// TwinCAT 3 PLC project POS_Temp_system
// ProgramVersion: 3.1.4022.3
// libraries:
//   CAA Types Extern, * (CAA Technical Workgroup)
//   Tc2_ControllerToolbox, * (Beckhoff Automation GmbH)
//   Tc2_Standard, * (Beckhoff Automation GmbH)
//   Tc2_System, * (Beckhoff Automation GmbH)
//   Tc2_Utilities, * (Beckhoff Automation GmbH)
//   Tc3_Module, * (Beckhoff Automation GmbH)
//   VisuSymbols,3.5.10.0,System
// project tree:
//   DUTs/ SeqState.TcTLEO
//   fbBLOCKS/ fbSensorNoise.TcPOU, FirstOrder.TcPOU
//   / GlobalTextList.TcGTLO, PlcTask.TcTTO, Visualization Manager.TcVMO (not stored)
//   GVLs/ GVL_IO.TcGVL
//   POUs/ fBDISCRETE_PID.TcPOU, MAIN.TcPOU
//   PROCESSES/ HEATER_PROCESS.TcPOU, SERVO_POS.TcPOU, TANKLEVEL.TcPOU
//   VISUs/ UserInterface.TcVIS
// real-time tasks:
//   TASK PlcTask: cycle T#10ms, priority 6, ADS port 350
//   TASK VISU_TASK: cycle T#200000us, priority 30, ADS port 351

CONFIGURATION POS_Temp_system
    RESOURCE PLC ON TwinCAT3
        TASK PlcTask(INTERVAL := T#10ms, PRIORITY := 6);
        PROGRAM MAIN WITH PlcTask : MAIN;
        PROGRAM SERVO_POS WITH PlcTask : SERVO_POS;
        PROGRAM HEATER_PROCESS WITH PlcTask : HEATER_PROCESS;
        PROGRAM TANKLEVEL WITH PlcTask : TANKLEVEL;
    END_RESOURCE
END_CONFIGURATION

// ---- DUTs/SeqState.TcTLEO
{attribute 'qualified_only'}
{attribute 'strict'}
TYPE SeqState :
(
	Ready,
	Fill_A,
	Fill_B,
	Heating,
	ToUnload,
	MovingToDrain,
	MovingToStart,
	Drain_1,
	Drain_2
	);
END_TYPE

// ---- GVLs/GVL_IO.TcGVL
{attribute 'qualified_only'}
VAR_GLOBAL
// Process parameters, variables	
	SetPoint_ServoX           :REAL;      // SetPoint X - axis
	SetPointHeater            :REAL;      // SetPoint Heater
	Output_ServoX             :REAL;      // X-axis Position
	Output_Heater             :REAL;      // Temperature Heater
	TankLevelSensor           :REAL;      // Tanklevel analogue sensor 
	ValveA, ValveB, ValveC    :BOOL;      // Valves
	xPushButton1              :BOOL;      // Used for test purposes 
	xPushButton2              :BOOL;      // Used for test purposes
	StartPr, StopPr           :BOOL;      // Start and Stop Process Buttons
	Level_S1,Level_S2,Level_S3:BOOL;      // Level Sensors (digital sensors)
    xGenCtrl_Error            :BOOL;      // General Error due SERVO or HEATER Control    
	Stirrer					  :BOOL;      //stirrer Set
	END_VAR

// ---- POUs/MAIN.TcPOU
PROGRAM MAIN
VAR
	PID_heater_enable: BOOL;  // PID Controller heater enabled ( Closed looop Control)
	PID_Servo_enable: BOOL := TRUE;   // PID Controller heater enabled ( Closed looop Control)
	pidServo  : fBDISCRETE_PID;
	pidHeater : fBDISCRETE_PID;
	States    : SeqState := SeqState.Ready;
	Cmd_Servo : R_TRIG;
	Cmd_Heater: R_TRIG;
	Cmd_ProdStart : R_TRIG;
	Cmd_ProdStop  : R_TRIG;
	HeaterON	  : BOOL;
	Rotation      : REAL;
	ToUnloadTimer : TON;
	TiMerToUnloadStart : BOOL;
	Counter : DINT;
	MoveTank : BOOL;
	StateString : STRING;
	
END_VAR

// Handling Buttons
Cmd_ProdStart(CLK:= GVL_IO.StartPr); 							// Start Process
Cmd_ProdStop(clk:=GVL_IO.StopPr);  								// Stop  Process
Cmd_Servo(clk:=MoveTank);    									// Servo Command button for testing
Cmd_Heater(clk:=GVL_IO.xPushButton2);   						// Heater Command button for testing
IF GVL_IO.Stirrer THEN     										// used to increas a counter
	Rotation := Rotation +5;									// used to rotate the stirrer in user interface
END_IF

IF Rotation = 359 THEN 											// if reached 360 degree reset
	Rotation := 0;
END_IF

ToUnloadTimer(IN := TiMerToUnloadStart ,PT := T#20S ); 			// timer to unload
// ================= START STATE SEQUENCE ======================
//
//   Your State machine program can be programmed here 
//          following an example
//

CASE States OF                       							// Sequence State ( ready, etc etc etc )
	SeqState.Ready:                  							// You can change the states if you want for your own convience
		StateString := 'Ready!';
		Counter := 0;											// sequence counter
		HeaterON := FALSE;
		IF GVL_IO.StartPr THEN 							// check if start button pressed
			States := SeqState.Fill_A;							// go to state Fill A
		END_IF
		
	SeqState.Fill_A:											// sequence state fill A
		StateString := 'Fill A';
		GVL_IO .ValveA:=TRUE;  									// open valve A				
		IF NOT GVL_IO.Level_S2 THEN 							// check if level reached s2
			GVL_IO.ValveA := FALSE;								//close valve A
			Counter := Counter + 1;									// increase counter after full cycle
			States := SeqState.Fill_B; 							// go to state Fill B
		END_IF
		
	SeqState.Fill_B:											// sequence state B
		StateString := 'Fill B';
		GVL_IO.SetPointHeater := 75; 							// set heater to 75
		HeaterON := TRUE;										//used in user interface to show heater lamp
		GVL_IO.Stirrer := TRUE; 								// set stirrer on 
		GVL_IO.ValveB := TRUE; 									// open valve B
		IF NOT GVL_IO.Level_S3 THEN 							// check if level s3 reached
			GVL_IO.ValveB := FALSE; 							// close valve B
			States := SeqState.ToUnload; 						// go to TOUnload state
		END_IF
		
	SeqState.ToUnload:											// sequence state TO Unload
		StateString := 'To Unload';
		TiMerToUnloadStart := TRUE;								// start ToUnloadTimer
		IF ToUnloadTimer.Q AND (GVL_IO.Output_Heater > 74.5 AND GVL_IO.Output_Heater < 76.5)  THEN									// if timer reached 20 sec
			TiMerToUnloadStart := FALSE;						// reset timer
			States := SeqState.MovingToDrain;					//go to MOving To drain state
		END_IF
	
	SeqState.MovingToDrain:										// sequence state moving to drain
		StateString := 'Move To Drain';
		MoveTank := TRUE;										// set move tank variable		
		GVL_IO.SetPoint_ServoX := 30;							// move tank to set point 30
		IF GVL_IO.Output_ServoX = 30 THEN						// if position reached
			MoveTank := FALSE;									// set move tank variable
			States := SeqState.Drain_1;							// go to drain 1 state
		END_IF
		
	SeqState.Drain_1:											// sequence state drain1
		StateString := 'Drain 1';
		GVL_IO.ValveC := TRUE;									//open valve c
		GVL_IO.SetPointHeater := 0;								//turn heater off
		HeaterON := FALSE;										// handle user interface variable
		IF GVL_IO.Level_S2 THEN									// if s2 level reached
			States := SeqState.Drain_2;							// go to drain 2 state
		END_IF
		
	SeqState.Drain_2:											//sequence state drain 2
		StateString := 'Drain 2';
		GVL_IO.Stirrer := FALSE;								// turn stirrer off
		IF GVL_IO.Level_S1 THEN									// if level s1 reached
			GVL_IO.ValveC := FALSE;								// close valve c 
			States := SeqState.MovingToStart;					// move to start position
		END_IF
	
	SeqState.MovingToStart: 									// sequence state move to start position
		StateString := 'Move To Start';
		MoveTank := TRUE;										// set move tank variable
		GVL_IO.SetPoint_ServoX := 0;							// set servo point to 0
		IF GVL_IO.Output_ServoX = 0 THEN						// if position 0 reached
			MoveTank := FALSE;									// set move tank variable
		IF Counter = 2 OR GVL_IO.StopPr THEN			
			States := SeqState.Ready;
		END_IF
		ELSE IF Counter < 2 AND NOT GVL_IO.StopPr THEN 
			States := SeqState.Fill_A;
		
		END_IF
		END_IF
	
		
		
		
//	
//
END_CASE
//
//

// ================ END STATE SEQUENCES=========================
// 


// =====   Executing the PID Controllers for  Position and Heater.   ===========
//==================================================================================
//
// *************  Servo with P- Controller only  **************
//
IF (MoveTank AND NOT GVL_IO.xGenCtrl_Error ) THEN
	pidServo.Setpoint:=GVL_IO.SetPoint_ServoX;  // Setpoint Servo // put in states
END_IF

pidServo.Kp:= 0.1;       //  Kp parameter
// pidServo.Ki:= xxx ; //  Ki parameter
// pidServo.Kd:= xxx ; //  Kd parameter 

pidServo.MV_max_sat:= 10;    // Maximum output PID to protect the Servo
pidServo.MV_min_sat:= -10;  // Minimum output PID    ,,     ,,
pidServo.xExt_Error:= Gvl_IO.xGenCtrl_Error;
//
pidServo.Yprocess:= LREAL_TO_REAL(GVL_IO.Output_ServoX);
//
pidServo(PID_enable:=PID_Servo_enable);  // Calling PID function Heater

// *************   Heater with P- Controller only   **********************
//
IF HeaterON THEN
   pidHeater.Setpoint:=GVL_IO.SetPointHeater;	
END_IF
IF HeaterON = FALSE THEN
	pidHeater.Setpoint := 0;
END_IF
pidHeater.Kp:= 1;         //  Kp parameter
// pidHeater.Ki:= xx ;    //  Ki parameter     
// pidHeater.Kd:= xx ;    //  Kd parameter      
pidHeater.MV_max_sat:=150;   // Maximum output PID to protect the Heater
pidHeater.MV_min_sat:= -10;  // Minimum output PID ,,     ,,
// 
pidHeater.Yprocess:=GVL_IO.Output_Heater;

pidHeater(PID_enable:= PID_heater_enable);  // Calling PID function Servo

END_PROGRAM

// ---- POUs/fBDISCRETE_PID.TcPOU
FUNCTION_BLOCK fBDISCRETE_PID
VAR_INPUT
	Setpoint:REAL;         // SetPoint
    Kp:REAL;               // Kp  Proportional gain
	Ki:REAL;               // Ki  Integrated gain
	Kd:REAL;               // Kd  Derivative gain
	Nfilter:REAL;          // Lowpass Filter Coeff 
	Yprocess :REAL;        // Process Output
	PID_enable : BOOL;     // PId enable (closed loop )
	MV_max_sat : REAL;     // Maximum Saturation
	MV_min_sat : REAL;     // Minimum Saturation
	xExt_Error  :BOOL;     // External error 
END_VAR
VAR_OUTPUT
	MV_out: REAL;
	Inposition:BOOL;     //  4% Settled 
END_VAR
VAR
	T1:DWORD :=0;
	T2:DWORD;
	Perr, Perr1, Perr2 : REAL ;
	A,B,C : REAL;
	prevMV_out:REAL;
	Tsample:REAL;
END_VAR

//
IF T1 = 0 THEN
	MV_out:=0;     // no bias offset controller
END_IF

Tsample:=0.01;
T1:=REAL_TO_DWORD(Tsample);
Perr:= Setpoint - Yprocess; // Current error e[k]
//
// Constant Coefficients including the Parameters Kp , Ki, Kd and Tsample
//        Your PID Controller algorithm starts here
//
//
//
//
//   Mv_out:=                                  // PID Controller
//
MV_out:=  Kp * Perr;  // P-Controller

// Update  samples 
prevMV_out := MV_out; // prevMV_out = MV_out[k-1] 
Perr2 := Perr1;       // e[k-2]
Perr1 := Perr;        // e[k-1]

//  PID  is not Enabled 
IF NOT PID_enable THEN
	MV_Out:= Setpoint;
END_IF

//    PID  output saturation 
IF Mv_out < MV_min_sat THEN
	Mv_out:= MV_min_sat;
END_IF
IF Mv_out >  MV_max_sat THEN
	Mv_out:= MV_max_sat;
END_IF
//  PID Output = 0 on External Error <user defined>
IF xExt_Error THEN
	Mv_out:=0;
END_IF

END_FUNCTION_BLOCK

// ---- PROCESSES/SERVO_POS.TcPOU
PROGRAM SERVO_POS
VAR CONSTANT
	nTfOrder : USINT := 2;
	nNumOrder : USINT :=2;
	nDenOrder : USINT :=2;
END_VAR
VAR
	aNumArray    : ARRAY[0..nNumOrder] OF FLOAT; //numerator
	aDenArray    : ARRAY[0..nDenOrder] OF FLOAT; //denumerator
	aStructTfData: ARRAY[0..nTfOrder]  OF ST_CTRL_TRANSFERFUNCTION_1_DATA;
	eMode : E_CTRL_MODE;
	stParams : ST_CTRL_TRANSFERFUNCTION_1_PARAMS;
	eErrorId : E_CTRL_ERRORCODES;
	bError : BOOL;
	fbServoX_Tf : FB_CTRL_TRANSFERFUNCTION_1;
	bInit : BOOL := TRUE;
	bPosError:BOOL;
	Tf_Output : LREAL;
	Servo_ERR : R_TRIG;

END_VAR

// IA _Cs4  2019
// O.E Figaroa
// Transferfunction Servo Motor X s-domain
//              20
//  Gc =    -----------   [ Theta/u]
//           0.5s^2 + s 
//
//= = Discrete or z-domain with  Ts = 0.01 s = = 
//          short format
//        0.001987 z + 0.001974
// Gd =  ----------------------   with Ts=0.01 s
//        z^2 - 1.98 z + 0.9802       
// 
//// coefficients obtained by Matlab in long format:
//
// numz =  [0   0.001986733067553   0.001973532271096]     
// denz =  [1.000000000000000 -1.980198673306755   0.980198673306755]
// ==

//========================================
IF bInit THEN
// = numerator ===
aNumArray[0] := 0.001973532271096; 
aNumArray[1] := 0.001986733067553; 
aNumArray[2] := 0.000;
// = denumerator
aDenArray[0] := 0.980198673306755;
aDenArray[1] := -1.980198673306755;
aDenArray[2] := 1.0;
stParams.tTaskCycleTime := T#10MS;
stParams.tCtrlCycleTime := T#10MS;
stParams.nOrderOfTheTransferfunction := nTfOrder;
eMode := eCTRL_MODE_ACTIVE;
bInit := FALSE;
END_IF
stParams.pNumeratorArray_ADR := ADR(aNumArray);
stParams.nNumeratorArray_SIZEOF := SIZEOF(aNumArray);
stParams.pDenominatorArray_ADR := ADR(aDenArray);
stParams.nDenominatorArray_SIZEOF := SIZEOF(aDenArray);
stParams.pTransferfunction1Data_ADR := ADR(aStructTfData);
stParams.nTransferfunction1Data_SIZEOF := SIZEOF(aStructTfData);

// Execute TF 

fbServoX_Tf (fIn :=main.pidServo.MV_out,
eMode := eMode,
stParams := stParams,
fOut => Tf_Output,
eErrorId => eErrorId,
bError => bError);

GVL_IO.Output_ServoX:=LREAL_TO_REAL(fbServoX_Tf.fOut);	

Servo_ERR(CLK:=(ABS(GVL_IO.Output_ServoX) > 50),Q=>GVL_IO.xGenCtrl_Error);

END_PROGRAM

// ---- PROCESSES/HEATER_PROCESS.TcPOU
PROGRAM HEATER_PROCESS
VAR CONSTANT
	nTfOrder : USINT := 2;
	nNumOrder : USINT :=2;
	nDenOrder : USINT :=2;
END_VAR
VAR
	aNumArray    : ARRAY[0..nNumOrder] OF FLOAT; //numerator
	aDenArray    : ARRAY[0..nDenOrder] OF FLOAT; //denumerator
	aStructTfData: ARRAY[0..nTfOrder]  OF ST_CTRL_TRANSFERFUNCTION_1_DATA;
	eMode : E_CTRL_MODE;
	stParams : ST_CTRL_TRANSFERFUNCTION_1_PARAMS;
	eErrorId : E_CTRL_ERRORCODES;
	bError : BOOL;
	fbHeater_Tf : FB_CTRL_TRANSFERFUNCTION_1;
	bInit : BOOL := TRUE;
	Tf_In : FLOAT := 0;
	Setpoint_Heater :INT;
	Tf_Heater_Output : LREAL;

END_VAR

// IA _Cs4  2019
// O.E Figaroa
// Transferfunction Heater
//                  5
///  G(s)=  ---------------------    [ Temp / Temp ]
//          256 s^2 + 100 s + 5
//= = = = = = = = = = = = = = = = 
// Discrete transfer function
//
//
//          9.753E-07 z + 9.74E-07
// G(z)=  ----------------------
//          z^2 - 1.996 z + 0.9961
//
// Obtained coefficients in long formats due accuracy
//
// numerator =    1.0e-06 * [0   0.975292016341129   0.974022931328863]
// denumerator = [1.000000000000000  -1.996099420155170   0.996101369470118]

IF bInit THEN
// = numerator ===
aNumArray[0] := 0.974022931328863 * 1E-06;
aNumArray[1] := 0.975292016341129 * 1E-06;
aNumArray[2] := 0.000;
// = denumerator
aDenArray[0] := 0.996101369470118;
aDenArray[1] := -1.996099420155170;
aDenArray[2] := 1.00000;
stParams.tTaskCycleTime := T#10MS;
stParams.tCtrlCycleTime := T#10MS;
stParams.nOrderOfTheTransferfunction := nTfOrder;
eMode := eCTRL_MODE_ACTIVE;
bInit := FALSE;
END_IF
stParams.pNumeratorArray_ADR := ADR(aNumArray);
stParams.nNumeratorArray_SIZEOF := SIZEOF(aNumArray);
stParams.pDenominatorArray_ADR := ADR(aDenArray);
stParams.nDenominatorArray_SIZEOF := SIZEOF(aDenArray);
stParams.pTransferfunction1Data_ADR := ADR(aStructTfData);
stParams.nTransferfunction1Data_SIZEOF := SIZEOF(aStructTfData);
// Execute TF 
fbHeater_Tf (fIn := main.pidHeater.MV_out,
eMode := eMode,
stParams := stParams,
fOut => Tf_Heater_Output,
eErrorId => eErrorId,
bError => bError);
//
GVL_IO.Output_Heater:=LREAL_TO_REAL(fbHeater_Tf.fOut);
IF fbHeater_Tf.fOut <= 0 THEN
	GVL_IO.Output_Heater:=0;
END_IF

END_PROGRAM

// ---- PROCESSES/TANKLEVEL.TcPOU
PROGRAM TANKLEVEL
VAR CONSTANT
	L_S1:REAL :=  5.00 ;
	L_S2:REAL := 60.00 ;
	L_S3:REAL := 80.00 ;	
END_VAR

VAR
	Plant:FirstOrder;
	fbNoise : FB_CTRL_NOISE_GENERATOR ;
	fbNoiseParams : ST_CTRL_NOISE_GENERATOR_PARAMS ;
	noise_level : LREAL ;
	fill_ValveA,fill_ValveB,Drain_ValveC: BOOL;
	fbdelayOFF:TOF;
// ---	
    fbFill, fbDrain : R_TRIG;
	fbFillOff, fbDrainOff :F_TRIG;
	currConstTime: REAL := 15;
	spLevel : REAL:=0;

END_VAR

// Generate sensor noise
fbNoiseParams . tCtrlCycleTime := T#10MS ;
fbNoiseParams . tTaskCycleTime := T#10MS ;
fbNoiseParams . fAmplitude := 1.5 ;
fbNoise ( fManSyncValue := 1 , eMode := 2 , stParams := fbNoiseParams ) ;
noise_level := fbNoise.fOut ;
// Valves
Fill_ValveA := GVL_IO.ValveA ;
Fill_ValveB := GVL_IO.ValveB ;
Drain_ValveC := GVL_IO.ValveC ;

fbFill(clk := ( Fill_ValveA XOR Fill_ValveB ) AND NOT Drain_ValveC ) ;
fbFillOff(clk := Fill_ValveA XOR Fill_ValveB ) ;
fbDrain(clk := Drain_ValveC );
fbDrainOff(clk := Drain_ValveC );
fbdelayOFF(IN:=(GVL_IO.ValveA OR GVL_IO.ValveB OR GVL_IO.ValveC),PT:=T#1S);

IF fbFill.Q THEN
	spLevel:=150;
	currConstTime:=15;
END_IF
IF fbFillOff.Q THEN
	spLevel:=plant.fBOut;
	
END_IF
IF fbDrain.Q THEN
	currConstTime:=5;
    spLevel:=1;	
END_IF

IF fbDrainOff.Q THEN
	spLevel := GVL_IO.TankLevelSensor ;
END_IF

Plant(fBIn:= spLevel,Gain := 1,Tconstant := currConstTime);

GVL_IO.TankLevelSensor:=plant.fBOut;

IF (fbdelayOFF.Q) THEN
	GVL_IO.TankLevelSensor:=LREAL_TO_REAL(plant.fBOut +noise_level);
END_IF
GVL_IO.Level_S1:=TRUE;
GVL_IO.Level_S2:=TRUE;
GVL_IO.Level_S3:=TRUE;

IF GVL_IO.TankLevelSensor > L_S1 THEN
	GVL_IO.Level_S1:=FALSE;
END_IF
IF GVL_IO.TankLevelSensor > L_S2 THEN
	GVL_IO.Level_S2:=FALSE;
END_IF
IF GVL_IO.TankLevelSensor > L_S3 THEN
	GVL_IO.Level_S3:=FALSE;
END_IF

 //

END_PROGRAM

// ---- fbBLOCKS/FirstOrder.TcPOU
FUNCTION_BLOCK FirstOrder
VAR_INPUT
	Gain: REAL;
	Tconstant : REAL;
	fBIn   : REAL;
END_VAR
VAR_OUTPUT
	fBOut  : REAL;
END_VAR
VAR
	ssy, Sy   :REAL;
	Tsample: REAL := 0.01;
END_VAR

// Euler Emulation 1st Order with 0.01 sec sampletime.
sy := ( fBIn * Gain / Tconstant ) - ( fBOut / Tconstant ) ;
fBOut := fBout + ( sy * Tsample ) ;

END_FUNCTION_BLOCK

// ---- fbBLOCKS/fbSensorNoise.TcPOU
FUNCTION_BLOCK fbSensorNoise
VAR_INPUT
	noise_enable:BOOL;
END_VAR
VAR_OUTPUT
noise_level : REAL;	
END_VAR
VAR
	fBNoise:FB_CTRL_NOISE_GENERATOR;
	fbNoiseParams: ST_CTRL_NOISE_GENERATOR_PARAMS;
END_VAR

// Generate noise for Sensors ( simulation ) 
fbNoiseParams.tCtrlCycleTime := T#10MS ;
fbNoiseParams.tTaskCycleTime := T#10MS ;
fbNoiseParams.fAmplitude := 1.5 ;
//
noise_level:=0;
IF Noise_enable THEN
	fbNoise ( fManSyncValue := 1 , eMode := 2 , stParams := fbNoiseParams ) ;
END_IF
noise_level:=fbNoise.fOut;

END_FUNCTION_BLOCK

// ---- GlobalTextList.TcGTLO
TEXTLIST GlobalTextList
  249 = '%.1d'
  0 = '%.1f'
  112 = '%.2f'
  464 = '%s'
  306 = '%s.'
  293 = 'A'
  602 = 'B'
  392 = 'C'
  753 = 'Drain Position'
  741 = 'gh'
  33 = 'GVL_IO.Output_ServoX * 10'
  303 = 'H'
  242 = 'Heater'
  601 = 'Home'
  193 = 'Level%.2f'
  167 = 'Outlet'
  445 = 'Output Heater   %.2f'
  735 = 'Output PID  %.2f'
  160 = 'Output Servo   %.2f'
  940 = 'Overshoot'
  350 = 'Overshoot= 30'
  17 = 'PID-Enable'
  786 = 'PID-Enable Heater'
  168 = 'PID-Enable Servo'
  520 = 'Position %s'
  569 = 'Position & Temperature Controle In Batch Processing'
  524 = 'Position & Temperature Controle In Batch Processing , IA , Hussam Ayoub'
  468 = 'Position = 0'
  917 = 'Position = 30'
  409 = 'Position and Temperature Control in Batch Process'
  224 = 'Position and Temperature Control in Batch Processes'
  93 = 'Response %s'
  81 = 'Response X -axis %s'
  617 = 'Response X -axis:   %s'
  12 = 'Response Y -axis %s'
  134 = 'Response Y -axis:   %s'
  251 = 'S1'
  356 = 'S2'
  849 = 'S3'
  150 = 'Servo Error'
  621 = 'Servo Running CCW'
  147 = 'Setpoint %.2f'
  636 = 'SetPoint %s'
  401 = 'Setpoint Heater   %.2f'
  352 = 'Setpoint Servo   %.2f'
  368 = 'SetPoint: %d'
  75 = 'SetPoint: %s'
  637 = 'SP Heater cmd'
  808 = 'SP Servo cmd'
  628 = 'Start'
  469 = 'Start Position'
  127 = 'Stop'
  527 = 'Tank'
  652 = 'TANK'
  181 = 'Tanklevel Sensor:    %.2f'
END_TEXTLIST

// ---- VISUs/UserInterface.TcVIS
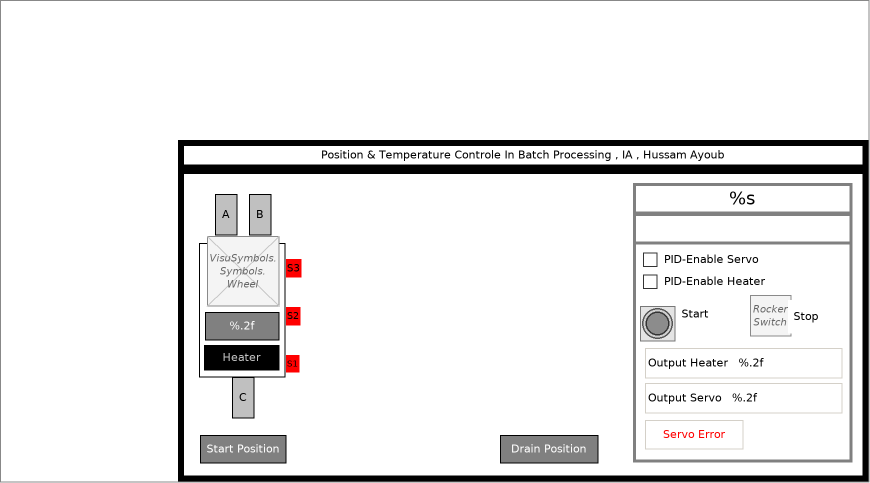
VISUALIZATION UserInterface  // 870x483
    Rectangle (178,168 690x313)
    Rectangle (633,239 219x223)
    Textfield (645,383 197x30), "Output Servo %.2f", text variable: GVL_IO.Output_ServoX
    Textfield (645,348 197x30), "Output Heater %.2f", text variable: GVL_IO.Output_Heater
    Rectangle (200,435 86x28), "Start Position"
    Rectangle (500,435 98x28), "Drain Position"
    Rectangle (199,243 86x134)
        p3560616238: GVL_IO.Output_ServoX * 10
    Textfield (633,213 219x31)
    Checkbox (641,270 123x23), "PID-Enable Heater", variable: MAIN.PID_heater_enable
    Checkbox (641,248 155x23), "PID-Enable Servo", variable: MAIN.PID_Servo_enable
    Textfield (645,420 98x29), "Servo Error", invisible if: NOT GVL_IO.xGenCtrl_Error
    Rectangle (215,194 22x41), "A", colour toggle: GVL_IO.ValveA
    Rectangle (249,194 22x41), "B", colour toggle: GVL_IO.ValveB
    Rectangle (232,377 22x41), "C", colour toggle: GVL_IO.ValveC
        p3560616238: GVL_IO.Output_ServoX * 10
    Rectangle (286,307 14x18), "S2", colour toggle: GVL_IO.Level_S2
        p3560616238: GVL_IO.Output_ServoX * 10
    Rectangle (286,259 15x18), "S3", colour toggle: GVL_IO.Level_S3
        p3560616238: GVL_IO.Output_ServoX * 10
    Rectangle (286,355 13x17), "S1", colour toggle: GVL_IO.Level_S1
        p3560616238: GVL_IO.Output_ServoX * 10
    Image (207,236 72x70), image: VisuSymbols.Symbols.Wheel
        p2858320360: MAIN.Rotation
        p3560616238: GVL_IO.Output_ServoX * 10
    Rectangle (204,345 75x25), "Heater", colour toggle: MAIN.HeaterON
        p3560616238: GVL_IO.Output_ServoX * 10
    RockerSwitch (750,295 41x41), variable: GVL_IO.StopPr, behaviour: TOGGLE, style: Switch-RockerSwitch-Gray
    Textfield (670,299 50x30), "Start"
    Textfield (788,300 36x33), "Stop"
    PushSwitch (640,297 35x53), variable: GVL_IO.StartPr, behaviour: TOGGLE, style: Switch-PushSwitch-Gray
    Textfield (633,183 219x31), "%s", text variable: MAIN.StateString
    Rectangle (178,140 690x30), "Position & Temperature Controle In Batch Processing , IA , Hussam Ayoub"
    Rectangle (205,312 74x28), "%.2f", text variable: GVL_IO.TankLevelSensor
        p3560616238: GVL_IO.Output_ServoX * 10
END_VISUALIZATION
